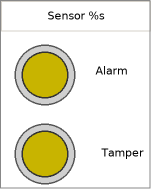
VISUALIZATION Sensor  // 151x189
VAR_IN_OUT
	stSensor		: ST_AlarmSensorHMI;
END_VAR
    Lamp1 (10,40 70x70), variable: stSensor.bAlarm, style: Lamp-Lamp1-Yellow
    Label (87,56 49x30), "Alarm"
    Textfield (1,1 150x30), "Sensor %s", text variable: stSensor.sName
    Lamp1 (10,119 70x70), variable: stSensor.bTamper, style: Lamp-Lamp1-Yellow
    Label (98,138 49x30), "Tamper"
END_VISUALIZATION

(* stored: Version 1.1.0.1, ProductVersion 3.1.4024.12
   Visu Sensor: Id {67e974ee-6017-429e-9dc8-95d3074c54e6} *)
